(*

Record performance data to influxDB and ANY SQL database
--------------------------------------------------------


* Objects

   Item List:
   
       This is body of item lists
	   
   Second Item:

      This is body of second items.
	  
	  
History
=====================

.. csv-table::
	:header: Rev., Date,Description
	
	0, 2023-01-10,Initial edition
	1, 2023-02-27,Add reStructuredText
	2, 2024-06-01,Add SQL database support
	  
*)

PROGRAM SampleProgram

VAR CONSTANT
	RECORD_DATA_MAX_INDEX: UDINT := 49999;
END_VAR

VAR
	
	// Initial
	initialized : BOOL;
	
	// Datetime utilities
	fbDtUtil : FB_DatetimeUtilities;

	// PLC System parameters
    fbGetCurTaskIdx  : GETCURTASKINDEX;
	test_timer :TON; // Inclese workload rate
	bExecuting :BOOL;
	j:UDINT := 0;
	target: UDINT := 5000;
	test_var:ULINT;
	
	process_timer :TON; // Process time

	// for InfluxDB

	// Record data buffer
	DatabaseThroughputRecordData 		:DatabaseThroughput;	// for insert dataset
	DatabaseThroughputRecordBuffer 		:ARRAY [0..DBLibParam.DATA_BUFFER_SIZE] OF DatabaseThroughput;

	fbThroughputRecorder_influxDB		:BufferedRecord(
												GVL.fbInfluxDBRecorder, 
												ADR(DatabaseThroughputRecordBuffer)
										);		// record controller

	// For SQL DB

	// Record data buffer
	DatabaseThroughputRecordData_SQL 		:DatabaseThroughput_SQL;	// for insert dataset
	DatabaseThroughputRecordBuffer_SQL 		:ARRAY [0..DBLibParam.DATA_BUFFER_SIZE] OF DatabaseThroughput_SQL;

	fbThroughputRecorder_SQLDB			:BufferedRecord(
												GVL.fbSQLRecorder, 
												ADR(DatabaseThroughputRecordBuffer_SQL)
										);		// record controller

END_VAR

(* Initialize*)
IF NOT initialized THEN
	// Influx DB
	fbThroughputRecorder_influxDB.set_buffer_info(
		struct_size := SIZEOF(DatabaseThroughputRecordBuffer[0]),
		buffer_size := SIZEOF(DatabaseThroughputRecordBuffer),
		structure_name := 'DatabaseThroughput'); // Measurement name
	fbThroughputRecorder_influxDB.SQL_parameters.table_name := 'DatabaseThroughput'; // Structure type name
	// SQL DB
	fbThroughputRecorder_SQLDB.set_buffer_info(
		struct_size := SIZEOF(DatabaseThroughputRecordBuffer_SQL[0]),
		buffer_size := SIZEOF(DatabaseThroughputRecordBuffer_SQL),
		structure_name := ''); // Measurement name
	fbThroughputRecorder_SQLDB.SQL_parameters.table_name := 'database_throughput';
	fbThroughputRecorder_SQLDB.SQL_parameters.add_column('datetime', E_ExpParameterType.Int64, SIZEOF(DatabaseThroughputRecordData_SQL.datetime));
	fbThroughputRecorder_SQLDB.SQL_parameters.add_column('db_insert_queue_count', E_ExpParameterType.Int32, SIZEOF(DatabaseThroughputRecordData_SQL.db_insert_queue_count));
	fbThroughputRecorder_SQLDB.SQL_parameters.add_column('current_index', E_ExpParameterType.Int32, SIZEOF(DatabaseThroughputRecordData_SQL.current_index));
	fbThroughputRecorder_SQLDB.SQL_parameters.add_column('next_index', E_ExpParameterType.Int32, SIZEOF(DatabaseThroughputRecordData_SQL.next_index));
	fbThroughputRecorder_SQLDB.SQL_parameters.add_column('buffer_usage', E_ExpParameterType.Float32, SIZEOF(DatabaseThroughputRecordData_SQL.buffer_usage));
	initialized := TRUE;
END_IF


fbDtUtil();


(*
	Database Throughput data insert buffer
*)


(* Data set here *)
// cyclic record > influxdb

// Tag Data
DatabaseThroughputRecordData.machine_id := 'machine-1';
DatabaseThroughputRecordData.job_id := 'db_throughput';
// Field data
DatabaseThroughputRecordData.db_insert_queue_count := GVL.fbInfluxDBRecorder.queue.queue_usage;
DatabaseThroughputRecordData.current_index := fbThroughputRecorder_influxDB.index;
DatabaseThroughputRecordData.next_index := fbThroughputRecorder_influxDB.next_index;
DatabaseThroughputRecordData.buffer_usage := fbThroughputRecorder_influxDB.buffer_usage;

(* Queue set *)
fbThroughputRecorder_influxDB.write(ADR(DatabaseThroughputRecordData));

// cyclic record > SQLdb
DatabaseThroughputRecordData_SQL.datetime := fbDtUtil.Filetime_To_UnixT(F_GetSystemTime());
DatabaseThroughputRecordData_SQL.db_insert_queue_count := GVL.fbSQLRecorder.queue.queue_usage;
DatabaseThroughputRecordData_SQL.current_index := fbThroughputRecorder_SQLDB.index;
DatabaseThroughputRecordData_SQL.next_index := fbThroughputRecorder_SQLDB.next_index;
DatabaseThroughputRecordData_SQL.buffer_usage := fbThroughputRecorder_SQLDB.buffer_usage;

fbThroughputRecorder_SQLDB.write(ADR(DatabaseThroughputRecordData_SQL));

END_PROGRAM

(* stored: Version 1.1.0.1, ProductVersion 3.1.4024.12
   POU SampleProgram: Id {54c36bd4-1835-4b4c-be1e-05e28c01780d}, SpecialFunc None *)
